INTERFACE IACPoint EXTENDS IACObject

METHOD AddEdge : BOOL
VAR_INPUT
	edge : IACEdge;
END_VAR
END_METHOD

PROPERTY ConnectionList : ARRAY [1..GCL.cEdgeMAX] OF IACEdge
GET
END_GET
END_PROPERTY

METHOD GetAllocatedEdge : IACEdge
VAR_INPUT
	paFunction : IPAProcessFunction;
END_VAR
END_METHOD

PROPERTY Parent : IACComponent
GET
END_GET
END_PROPERTY

END_INTERFACE

(* stored: Version 1.1.0.1, ProductVersion 3.1.4020.12
   Itf IACPoint: Id {5757c0fc-3675-430f-b1d8-f13cc716bbf3}
   Method AddEdge: Id {a39e5a6a-5cf1-4847-bb5d-865a8f7ee40b}
   Property ConnectionList: Id {5652df52-ca8d-4bd3-81e2-5c4f954d1764}
   Get Get: Id {b2c227b2-863e-439f-9cea-b4405f043d8f}
   Method GetAllocatedEdge: Id {69470acd-105a-4d11-8a4f-7936d42703b2}
   Property Parent: Id {e4a78408-b62c-4f5e-a4a4-de7990f1c96f}
   Get Get: Id {da73d826-06d7-444a-8121-494d96625d35} *)
